FUNCTION_BLOCK OpticalSensor IMPLEMENTS ITF_BinarySensor
VAR_INPUT
END_VAR
VAR_OUTPUT
END_VAR
VAR
	//Hardware
	DI_WPLight AT %I* : BOOL;
END_VAR

PROPERTY Value : BOOL
GET
Value := DI_WPLight;
END_GET
END_PROPERTY

END_FUNCTION_BLOCK

(* stored: Version 1.1.0.1
   POU OpticalSensor: Id {ea8f7113-9a03-4926-8603-058b2d122585}, SpecialFunc None
   Property Value: Id {5b23ff69-c222-46bf-a742-79a419134b98}
   Get Get: Id {370d13e6-f0fd-44aa-8fdb-6ce4fe4e67ea} *)
